(* CODESYS project xlh_ha_client_00_01.project
   Author: CODESYS Development GmbH
   Title: MQTT Client SL Example
   Company: CODESYS

Project tree, tasks and I/O mapping:
  Device : CODESYS Control for Raspberry Pi 64 SL, CODESYS, order no. 2302000009, version 4.12.0.0
    application app
      libraries: Standard, 3.5.18.0 (System); StringUtils, 3.5.20.0 (System); VisuDialogs, * (System); Web Socket Client SL, 1.12.0.0 (CODESYS); Net Base Services, * (3S - Smart Software Solutions GmbH); MQTT Client SL, 1.12.0.0 (CODESYS); Util, 3.5.21.0 (System); String Functions, * (CODESYS); SysTimeRtc, * (System); SysTime, 3.5.17.0 (System); CmpIecTask, * (System)
      task MainTask (cyclic, interval t#20ms, priority 1) calls LOCAL_TIME_AND_TIME_ZONE, TASK_INFO, io, MAIN
      program MAIN [ST]
      program io [ST]
      IoT/
        DEVICES/
          function block _100_FB_DEVICE [ST]: subscriber, publisher, pMqttClient, startup, sMqttTopicBase, newMessage, statusUpdate
          function block _200_FB_DEVICE_SHELLY_BASE [ST]: statusUpdate, startup, newMessage
          function block _202_FB_DEVICE_SHELLY_1PM_TEMP [ST]: newMessage
          interface IDevice
          interface IDeviceZigbee2Mqtt
          interface IDeviceShelly
          function block _201_FB_DEVICE_SHELLY_1PM_PLUG [ST]: publisher, newMessage
        MQTT_Client/
          function TERMINATE_STRING [ST]
          function block FB_MQTT_CLIENT [ST]: pMqttClient
          function GET_VALUE_FROM_MSG [ST]
          function GET_REAL_FROM_VALUE [ST]
          function GET_BOOL_FROM_VALUE [ST]
          function GET_INT_FROM_VALUE [ST]
          function GET_STRING_FROM_VALUE [ST]
        global variables GC
        program TASK_INFO [ST]
        program LOCAL_TIME_AND_TIME_ZONE [ST]
    SoftMotion General Axis Pool
    GPIOs_A_B : GPIOs A/B, CODESYS, version 4.18.0.0
        unmapped channels: digital inputs (GPIO0..GPIO31), digital outputs (GPIO0..GPIO31)
    Onewire
    Camera device
      <Empty>
    SPI
    I²C
  text list GlobalTextList
  5ce3da45-db07-42e7-a21c-a00fff4ed8f6|C:\Users\a.werner\Documents\background.jpg
*)

// Device/app/IoT/GC
{attribute 'qualified_only'}
VAR_GLOBAL CONSTANT
	//STRING_SIZE: INT := 255;
	STRING_SIZE_TOPIC: INT := 1024;
	STRING_SIZE_MESSAGE_RCV: INT := 2048;
END_VAR

// Device/app/IoT/LOCAL_TIME_AND_TIME_ZONE
PROGRAM LOCAL_TIME_AND_TIME_ZONE
VAR_OUTPUT
	stUTC_Timestamp : SysTime;
	stCTE_Timestamp : SysTime;
	stJoinedTimestamp : SysTime;
	stCombinedTimestamp : SysTime;
	uiYear : YEAR; (* 1970..2106 *)
    uiMonth : MONTH;
    uiDay : DAY;
    uiHour : UINT;
    uiMinute : UINT;
    uiSecond : UINT;
    uiMilliseconds : MILLISECOND;
    eWeekday : WEEKDAY;
    datDate : DATE;
    todTime : TIME_OF_DAY;
	eError : Util.ERROR;
	xLeapYear : BOOL;
END_VAR
VAR CONSTANT
    /// Coordinated Universal Time
    gc_tzTimeZoneUTC : TimeZone := (asgPeriod := [(sName:='UTC')]);

    /// Central Europe Time
    gc_tzTimeZoneCET : TimeZone :=
    (
        iBias := 60 (* T#1M => minutes *),
        asgPeriod := [
        ( (* (CEST -> CET) - Last Sunday in Oktober at 03:00:00.000 (CEST) *)
            sName:='CET',
            dtDate := (uiMonth := 10, eWeekday := WEEKDAY.SUNDAY, uiDay := 5, uiHour := 3)
        ),( (* (CET -> CEST) - Last Sunday in March at 02:00:00.000 (CET) *)
            sName := 'CEST',
            dtDate := (uiMonth := 3, eWeekday := WEEKDAY.SUNDAY, uiDay := 5, uiHour := 2),
            iBias := 60 (* T#1M => minutes *)
        )]
    );
END_VAR

SysTimeRtcHighResGet(pTimestamp := stUTC_Timestamp);
// Conversion from UTC timestamp (e.g. from SysTimeRtcHighResGet) to the current period and the local date and time related to the TimeZone parameter.
stCTE_Timestamp := Util.LocalDateTime(	tzTimeZone := gc_tzTimeZoneCET, 
										uliDateTime := stUTC_Timestamp,
										eErrorID => eError);

// Splitting a timestamp into the components of a point in time.
eError := Util.SplitDateTime(	uliDateTime := stCTE_Timestamp,
				uiYear => uiYear,
				uiMonth =>  uiMonth,
				uiDay => uiDay,
				uiHour => uiHour,
				uiMinute => uiMinute,
				uiSecond =>  uiSecond,
				uiMilliseconds => uiMilliseconds,
				eWeekday => eWeekday);

// Joining the components of a point in time to a timestamp (UTC). 
stJoinedTimestamp :=  Util.JoinDateTime( 	uiYear := uiYear,
									uiMonth :=  uiMonth,
									uiDay := uiDay,
									uiHour := uiHour,
									uiMinute := uiMinute,
									uiSecond :=  uiSecond,
									uiMilliseconds := uiMilliseconds);
									
// Separates a timestamp in its IEC data typed parts.
 Util.SeparateDateTime(	uliDateTime := stCTE_Timestamp,
    				eWeekDay => eWeekDay,
    				datDate => datDate,
    				todTime => todTime);
					
// Combines the IEC data typed parts to a timestamp.
stCombinedTimestamp := Util.CombineDateTime(	datDate := datDate, 
												todTime := todTime, 
												eErrorID => eError);
						
// Calculates the appropriate value of the WEEKDAY enum that matches the parameter datDate.
eWeekday := Util.DayOfWeek(	datDate := datDate, 
							eErrorID => eError);

// Checks whether the year (uiYear) passed represents a leap year.					
xLeapYear := Util.IsLeapYear(	uiYear := uiYear,
								eErrorID => eError);

END_PROGRAM

// Device/app/IoT/TASK_INFO
PROGRAM TASK_INFO
VAR
    Result: CmpIecTask.RTS_IEC_RESULT;
    hCurrentTask : CmpIecTask.RTS_IEC_HANDLE;
    pCurrentTaskInfo: POINTER TO Task_Info2;
    stCurrentTaskInfo: Task_Info2;
END_VAR
VAR_OUTPUT
	rCycleTime: REAL;
	rInterval: REAL;
	rCycleTimeUs: REAL;
	rJitterUs: REAL;
	rJitterOffsetInterwalUs: REAL;
END_VAR

// https://content.helpme-codesys.com/en/libs/CmpIecTask/Current/index.html
// https://forge.codesys.com/forge/talk/Engineering/thread/b7e9b2b353/
// https://medium.com/@sean.gongz/how-to-get-current-task-actual-cycle-time-in-codesys-267384bcd3b7

hCurrentTask := IecTaskGetCurrent(pResult:=ADR(Result));
pCurrentTaskInfo := IecTaskGetInfo3(hIecTask:=hCurrentTask, pResult:=ADR(Result));
stCurrentTaskInfo := pCurrentTaskInfo^;

rCycleTimeUs := TO_REAL(TO_DINT(stCurrentTaskInfo.dwInterval) + stCurrentTaskInfo.iJitter);
rInterval := TO_REAL(stCurrentTaskInfo.dwInterval);
rJitterUs := TO_REAL(stCurrentTaskInfo.iJitter);
rJitterOffsetInterwalUs := rInterval + rJitterUs;
rCycleTime := rCycleTimeUs / 1000000.0;

END_PROGRAM

// Device/app/io
PROGRAM io
VAR_INPUT
	fbShellyPlug1: _201_FB_DEVICE_SHELLY_1PM_PLUG;
	fbShellyPlug2: _201_FB_DEVICE_SHELLY_1PM_PLUG;
	fbShellyPm1: _202_FB_DEVICE_SHELLY_1PM_TEMP;
END_VAR
VAR
	_bStartup: BOOL := TRUE;
	_aIoClients: ARRAY [0..(iNR_OF_IO_CLIENTS-1)] OF POINTER TO _100_FB_DEVICE;
	_fbMqttClient: FB_MQTT_CLIENT;
	_iI: INT;
	//
	_bDummy: BOOL;
END_VAR
VAR CONSTANT
	iNR_OF_IO_CLIENTS: INT := 20;
END_VAR

IF _bStartup THEN
	_bStartup := FALSE;
	
	fbShellyPlug1.sMqttTopicBase := 'shellyplug-81';
	fbShellyPlug2.sMqttTopicBase := 'shellyplug-82';
	fbShellyPm1.sMqttTopicBase := 'shellyplus-51';
	
	_aIoClients[_iI] := ADR(fbShellyPlug1); _iI := _iI + 1;
	_aIoClients[_iI] := ADR(fbShellyPlug2); _iI := _iI + 1;
	_aIoClients[_iI] := ADR(fbShellyPm1); _iI := _iI + 1;
	
	FOR _iI := 0 TO (iNR_OF_IO_CLIENTS-1) BY 1 DO
		IF (_aIoClients[_iI] > 16#0) THEN
			_aIoClients[_iI]^.pMqttClient := ADR(_fbMqttClient);
			_aIoClients[_iI]^.startup();	
		END_IF
	END_FOR	
	
	_fbMqttClient.bEnable := TRUE;
END_IF

_fbMqttClient();

FOR _iI := 0 TO (iNR_OF_IO_CLIENTS-1) BY 1 DO
	IF (_aIoClients[_iI] >16#0) THEN
		_aIoClients[_iI]^();	
	END_IF
END_FOR

_bDummy := _fbMqttClient.bConnected;

END_PROGRAM

// Device/app/IoT/DEVICES/_201_FB_DEVICE_SHELLY_1PM_PLUG
FUNCTION_BLOCK _201_FB_DEVICE_SHELLY_1PM_PLUG EXTENDS _200_FB_DEVICE_SHELLY_BASE
VAR_INPUT
	bRelais: BOOL;
END_VAR
VAR_OUTPUT
	bRelaisState: BOOL;
	rVoltage: REAL;
	rCurrent: REAL;
	rPower: REAL;
END_VAR
VAR
	//
	_fbRtRelais: R_TRIG;
	_fbFtRelais: F_tRIG;
	_fbTonDiffRelaisState: TON;
END_VAR
VAR CONSTANT
	_tACTION_TIME_NOT_EQUAL: TIME := T#500MS;
END_VAR

SUPER^();

METHOD publisher : BOOL
VAR_INPUT
END_VAR

VAR
	bPublish: BOOL;
END_VAR
THIS^._fbTonDiffRelaisState(IN:=((THIS^.bRelais <> THIS^.bRelaisState) AND NOT _fbTonDiffRelaisState.Q), PT:=THIS^._tACTION_TIME_NOT_EQUAL);
THIS^._fbRtRelais(CLK:=THIS^.bRelais);
THIS^._fbFtRelais(CLK:=THIS^.bRelais);
bPublish := _fbTonDiffRelaisState.Q OR _fbRtRelais.Q OR _fbFtRelais.Q;

IF bPublish THEN
	THIS^._fbMqttPublisher.xExecute := TRUE;
	THIS^._sPublishMessage := '{"id":1, "src":"';
	THIS^._sPublishMessage := CONCAT(THIS^._sPublishMessage, THIS^._sMqttTopicBase);
	THIS^._sPublishMessage := CONCAT(THIS^._sPublishMessage, '/relais", "method":"Switch.Set", "params":{"id":0, "on":');
	IF THIS^.bRelais THEN
		THIS^._sPublishMessage := CONCAT(THIS^._sPublishMessage, 'true}}');
	ELSE
		THIS^._sPublishMessage := CONCAT(THIS^._sPublishMessage, 'false}}');
	END_IF
END_IF

SUPER^.publisher();

// '{"id":1, "src":"shellyplus-51/status", "method":"Shelly.GetStatus"}'
//{"id":1, "src":"shellyplus-51/relais", "method":"Switch.Set", "params":{"id":0, "on":true}}
END_METHOD

METHOD newMessage : BOOL
VAR_INPUT
	
END_VAR
VAR

	
END_VAR
SUPER^.newMessage();
IF (_fbMqttSubscriber.wsLastTopic = _wsMqttTopicEvent) OR
   (_fbMqttSubscriber.wsLastTopic = _wsMqttTopicStatus) THEN
	bRelaisState := GET_BOOL_FROM_VALUE(bRelaisState, GET_VALUE_FROM_MSG('output', ADR(_sSubscribedMessage)));
	rVoltage := GET_REAL_FROM_VALUE(rVoltage, GET_VALUE_FROM_MSG('voltage', ADR(_sSubscribedMessage)));
	rCurrent := GET_REAL_FROM_VALUE(rCurrent, GET_VALUE_FROM_MSG('current', ADR(_sSubscribedMessage)));
	rPower := GET_REAL_FROM_VALUE(rPower, GET_VALUE_FROM_MSG('apower', ADR(_sSubscribedMessage)));
		
END_IF
IF (_fbMqttSubscriber.wsLastTopic = _wsMqttTopicStatus) THEN
	sSsid := GET_STRING_FROM_VALUE(sSsid, GET_VALUE_FROM_MSG('ssid', ADR(_sSubscribedMessage)));
	sMacId := GET_STRING_FROM_VALUE(sSsid, GET_VALUE_FROM_MSG('bssid', ADR(_sSubscribedMessage)));	
END_IF
END_METHOD

END_FUNCTION_BLOCK

// Device/app/IoT/DEVICES/_200_FB_DEVICE_SHELLY_BASE
FUNCTION_BLOCK _200_FB_DEVICE_SHELLY_BASE EXTENDS _100_FB_DEVICE IMPLEMENTS IDeviceShelly
VAR_INPUT
END_VAR
VAR_OUTPUT
	rTemperaturePcb: REAL;
	sSsid: STRING(255);
	sMacId: STRING(255);
	iRssi: INT;
END_VAR
VAR
	//
	_wsMqttTopicEvent: WSTRING(GC.STRING_SIZE_TOPIC) := "shellyplus-51/status/rpc";
	_wsMqttTopicStatus: WSTRING(GC.STRING_SIZE_TOPIC) := "shellyplus-51/status/rpc";
	_rTimer: REAL := 0.0;
END_VAR
VAR CONSTANT
	_rREFRESH_TIME: REAL := 300.0;
END_VAR

SUPER^();

_rTimer := LIMIT(0.0, _rTimer + TASK_INFO.rCycleTime, 99999.0);
IF _rTimer >= _rREFRESH_TIME THEN
	_rTimer := 0.0;
	statusUpdate();
END_IF

METHOD statusUpdate : BOOL
VAR_INPUT
END_VAR

VAR
END_VAR
SUPER^.statusUpdate();

THIS^._fbMqttPublisher.xExecute := TRUE;
THIS^._sPublishMessage := '{"id":1, "src":"';
THIS^._sPublishMessage := CONCAT(THIS^._sPublishMessage, THIS^._sMqttTopicBase);
THIS^._sPublishMessage := CONCAT(THIS^._sPublishMessage, '/status", "method":"Shelly.GetStatus"}');

// '{"id":1, "src":"shellyplus-51/status", "method":"Shelly.GetStatus"}'
END_METHOD

METHOD startup : BOOL
VAR_INPUT
END_VAR

VAR
END_VAR
SUPER^.startup();

_wsMqttTopicEvent := "";
Stu.StrConcatW(pstFrom:=ADR(_wsMqttTopicBase), pstTo:=ADR(_wsMqttTopicEvent), iBufferSize:=GC.STRING_SIZE_TOPIC);
Stu.StrConcatW(pstFrom:=ADR("/events/rpc"), pstTo:=ADR(_wsMqttTopicEvent), iBufferSize:=GC.STRING_SIZE_TOPIC);
		
_wsMqttTopicStatus := "";
Stu.StrConcatW(pstFrom:=ADR(_wsMqttTopicBase), pstTo:=ADR(_wsMqttTopicStatus), iBufferSize:=GC.STRING_SIZE_TOPIC);
Stu.StrConcatW(pstFrom:=ADR("/status/rpc"), pstTo:=ADR(_wsMqttTopicStatus), iBufferSize:=GC.STRING_SIZE_TOPIC);
END_METHOD

METHOD newMessage : BOOL
VAR_INPUT
	
END_VAR
VAR

	
END_VAR
SUPER^.newMessage();
IF (_fbMqttSubscriber.wsLastTopic = _wsMqttTopicEvent) OR
   (_fbMqttSubscriber.wsLastTopic = _wsMqttTopicStatus) THEN
   rTemperaturePcb := GET_REAL_FROM_VALUE(rTemperaturePcb, GET_VALUE_FROM_MSG('temperature":{"tC', ADR(_sSubscribedMessage)));
	iRssi := GET_INT_FROM_VALUE(iRssi, GET_VALUE_FROM_MSG('rssi', ADR(_sSubscribedMessage)));	
END_IF
IF (_fbMqttSubscriber.wsLastTopic = _wsMqttTopicStatus) THEN
	sSsid := GET_STRING_FROM_VALUE(sSsid, GET_VALUE_FROM_MSG('ssid', ADR(_sSubscribedMessage)));
	sMacId := GET_STRING_FROM_VALUE(sSsid, GET_VALUE_FROM_MSG('bssid', ADR(_sSubscribedMessage)));	
END_IF
END_METHOD

END_FUNCTION_BLOCK

// Device/app/IoT/DEVICES/_100_FB_DEVICE
FUNCTION_BLOCK _100_FB_DEVICE IMPLEMENTS IDevice
VAR
	_pMqttClient: POINTER TO FB_MQTT_CLIENT;
	_wsMqttTopicBase: WSTRING(GC.STRING_SIZE_TOPIC);
	_sMqttTopicBase: STRING(255);
	//
	_fbRtMqttClientConnected: R_TRIG;
	_fbFtMqttClientConnected: F_TRIG;
	_fbRtMqttSubscriberActive: R_TRIG;
	_fbFtMqttSubscriberActive: F_TRIG;
	_fbRtError: R_TRIG;
	_fbTonConnect: TON;
	_fbTonDisconnect: TON;
	_fbMqttSubscriber : MQTT.MQTTSubscribe;
	_wsSubcribedTopicFilter : WSTRING(GC.STRING_SIZE_TOPIC);
	_sSubscribedMessage : STRING(GC.STRING_SIZE_MESSAGE_RCV);	
	_fbMqttPublisher : MQTT.MQTTPublish;
	_wsPublishTopic : WSTRING(GC.STRING_SIZE_TOPIC);
	_sPublishMessage : STRING(255);
	//
	_todMessageUpdate: TIME_OF_DAY;
	//
	_bDummy: BOOL;
	_iDummyCtr: INT;
	_sDummy: STRING(GC.STRING_SIZE_MESSAGE_RCV);
	_wsDummy: WSTRING(GC.STRING_SIZE_TOPIC);
END_VAR

(*
Optimierung:
- Queue für Verarbeitung ausgehender Nachrichten
- Interface
- REAL mit LReal ersetzen
*)

THIS^.subscriber();
THIS^.publisher();

METHOD subscriber : BOOL
VAR_INPUT
END_VAR
THIS^._fbRtMqttClientConnected(CLK:=THIS^._pMqttClient^.bConnected);
THIS^._fbFtMqttClientConnected(CLK:=THIS^._pMqttClient^.bConnected);
THIS^._fbRtError(CLK:=THIS^._pMqttClient^.bError);
IF THIS^._fbRtMqttClientConnected.Q THEN
	THIS^._fbMqttSubscriber.xEnable := TRUE;
END_IF
IF THIS^._fbRtError.Q OR THIS^._fbFtMqttClientConnected.Q THEN
	THIS^._fbMqttSubscriber.xEnable := FALSE;
END_IF
THIS^._fbTonDisconnect.IN := THIS^._pMqttClient^.bConnected AND THIS^._fbMqttSubscriber.xEnable AND NOT THIS^._fbMqttSubscriber.xBusy;
THIS^._fbTonDisconnect(PT:=T#3000MS);
IF THIS^._fbTonDisconnect.Q THEN
	THIS^._fbMqttSubscriber.xEnable := FALSE;
END_IF
THIS^._fbTonConnect.IN := THIS^._pMqttClient^.bConnected AND NOT THIS^._fbMqttSubscriber.xEnable;
THIS^._fbTonConnect(PT:=T#500MS);
IF THIS^._fbTonConnect.Q THEN
	THIS^._fbMqttSubscriber.xEnable := TRUE;
END_IF

THIS^._fbMqttSubscriber(mqttClient:=THIS^._pMqttClient^.fbMqttClient,
				wsTopicFilter:=THIS^._wsSubcribedTopicFilter,
		        pbPayload:=ADR(THIS^._sSubscribedMessage),
				udiMaxPayloadSize:=SIZEOF(THIS^._sSubscribedMessage));
TERMINATE_STRING(psIn:=ADR(THIS^._sSubscribedMessage), THIS^._fbMqttSubscriber.udiPayloadSize);

IF THIS^._fbMqttSubscriber.xReceived THEN
	THIS^.newMessage();
END_IF 

THIS^._fbRtMqttSubscriberActive(CLK:=THIS^._fbMqttSubscriber.xSubscribeActive);
THIS^._fbFtMqttSubscriberActive(CLK:=THIS^._fbMqttSubscriber.xSubscribeActive);
IF THIS^._fbRtMqttSubscriberActive.Q THEN
	THIS^.statusUpdate();
END_IF
			
_bDummy := THIS^._fbMqttSubscriber.xEnable;				
_bDummy := THIS^._fbMqttSubscriber.xDone;
_bDummy := THIS^._fbMqttSubscriber.xBusy;
_bDummy := THIS^._fbMqttSubscriber.xError;
_bDummy := THIS^._fbMqttSubscriber.xSubscribeActive;
_wsDummy := THIS^._fbMqttSubscriber.wsLastTopic;
_sDummy := THIS^._sSubscribedMessage;
END_METHOD

METHOD publisher : BOOL
VAR_INPUT
END_VAR
THIS^._fbMqttPublisher(mqttClient:=_pMqttClient^.fbMqttClient, 	 
                       wsTopicName:=_wsPublishTopic,
                       udiTimeOut:=10000,
                       pbPayload:=ADR(_sPublishMessage),
	                   udiPayloadSize:=DINT_TO_UDINT(Stu.StrLenA(ADR(_sPublishMessage))));

(*
// Send Counter
IF _fbMqttPublisher.xBusy THEN
	_iDummyCtr := _iDummyCtr + 1;
END_IF
*)

THIS^._fbMqttPublisher.xExecute := FALSE;   

_bDummy := _fbMqttPublisher.xDone;
_bDummy := _fbMqttPublisher.xBusy;
_bDummy := _fbMqttPublisher.xError;
_wsDummy := _wsPublishTopic;
_sDummy := _sPublishMessage;
END_METHOD

PROPERTY pMqttClient : POINTER TO FB_MQTT_CLIENT
GET
pMqttClient := THIS^._pMqttClient;
END_GET
SET
THIS^._pMqttClient := pMqttClient;
END_SET
END_PROPERTY

METHOD startup : BOOL
VAR_INPUT
END_VAR

VAR
END_VAR
_wsMqttTopicBase := STRING_TO_WSTRING(_sMqttTopicBase);

_wsPublishTopic := "";
Stu.StrConcatW(pstFrom:=ADR(_wsMqttTopicBase), pstTo:=ADR(_wsPublishTopic), iBufferSize:=GC.STRING_SIZE_TOPIC);
Stu.StrConcatW(pstFrom:=ADR("/rpc"), pstTo:=ADR(_wsPublishTopic), iBufferSize:=GC.STRING_SIZE_TOPIC);

_wsSubcribedTopicFilter := "";
Stu.StrConcatW(pstFrom:=ADR(_wsMqttTopicBase), pstTo:=ADR(_wsSubcribedTopicFilter), iBufferSize:=GC.STRING_SIZE_TOPIC);
Stu.StrConcatW(pstFrom:=ADR("/#"), pstTo:=ADR(_wsSubcribedTopicFilter), iBufferSize:=GC.STRING_SIZE_TOPIC);
END_METHOD

PROPERTY PUBLIC sMqttTopicBase : STRING(255)
SET
THIS^._sMqttTopicBase := sMqttTopicBase;
END_SET
GET
sMqttTopicBase := THIS^._sMqttTopicBase;
END_GET
END_PROPERTY

METHOD newMessage : BOOL
VAR_INPUT
	
END_VAR
VAR

	
END_VAR
THIS^._todMessageUpdate := LOCAL_TIME_AND_TIME_ZONE.todTime;
END_METHOD

METHOD statusUpdate : BOOL
VAR_INPUT
END_VAR

VAR
END_VAR
END_METHOD

END_FUNCTION_BLOCK

// Device/app/IoT/DEVICES/IDevice
INTERFACE IDevice

END_INTERFACE

// Device/app/IoT/MQTT_Client/FB_MQTT_CLIENT
FUNCTION_BLOCK FB_MQTT_CLIENT
VAR_INPUT
	bEnable: BOOL;
	sHostname: STRING(255) := 'localhost';	
	sClientId: STRING(255) := 'xLH_mqtt_codesys';	
END_VAR
VAR_OUTPUT
	bConnected: BOOL;
	bError: BOOL;
	fbMqttClient : MQTT.MQTTClient := (uiPort:=1883, eMQTTVersion:=MQTT.MQTT_VERSION.V3_1_1, eCommunicationMode:= MQTT.COMMUNICATION_MODE.TCP);
END_VAR
VAR
	_refMqttClient: REFERENCE TO MQTT.MQTTClient;
	_bStartup: BOOL := TRUE;
END_VAR

IF _bStartup THEN
	_bStartup := FALSE;
	_refMqttClient REF= fbMqttClient;
END_IF
fbMqttClient.xEnable := bEnable AND NOT fbMqttClient.xError;
fbMqttClient.sClientId := sClientId;
fbMqttClient(sHostname:=sHostname);
bConnected := fbMqttClient.xConnectedToBroker;
bError := fbMqttClient.xError;

PROPERTY pMqttClient : POINTER TO FB_MQTT_CLIENT
GET
pMqttClient := ADR(THIS^.fbMqttClient);
END_GET
END_PROPERTY

END_FUNCTION_BLOCK

// Device/app/IoT/MQTT_Client/TERMINATE_STRING
// Terminates the STRING psIn at position udiLength
FUNCTION TERMINATE_STRING : BOOL
VAR_INPUT
	psIn : POINTER TO BYTE; // Pointer to STRING
	udiLength : UDINT; // Length of psIn
END_VAR
VAR
END_VAR

psIn[udiLength] := 0;
TERMINATE_STRING := TRUE;

END_FUNCTION

// Device/app/IoT/DEVICES/IDeviceShelly
INTERFACE IDeviceShelly

END_INTERFACE

// Device/app/IoT/MQTT_Client/GET_REAL_FROM_VALUE
FUNCTION GET_REAL_FROM_VALUE: REAL;
VAR_INPUT
	rValue: REAL;
	sValue: STRING(255);
END_VAR

IF sValue <> '' THEN
	rValue := STRING_TO_REAL(sValue);
END_IF
GET_REAL_FROM_VALUE := rValue;

END_FUNCTION

// Device/app/IoT/MQTT_Client/GET_VALUE_FROM_MSG
FUNCTION GET_VALUE_FROM_MSG: STRING(255)
VAR_INPUT
	sKey: STRING(255);
	pSubscribedMessage: POINTER TO STRING(GC.STRING_SIZE_MESSAGE_RCV);
END_VAR
VAR
	iStrFindPos1: INT;
	iStrFindPos2: INT;
	sMessage : STRING(255);
	sValue : STRING(255);
END_VAR

sKey := CONCAT(CONCAT('"', sKey), '":'); 		

iStrFindPos1 := MAX(0, Stu.StrFindA(pst1:=pSubscribedMessage, pst2:=ADR(sKey), uiSearchStart:=0));
Stu.StrCpyA(pBuffer:=ADR(sMessage), 
			iBufferSize:=SIZEOF(sMessage)-50, 
			pStr:=pSubscribedMessage+INT_TO_DWORD(iStrFindPos1));  

iStrFindPos1 := MAX(0, Stu.StrFindA(pst1:=ADR(sMessage), 
                                    pst2:=ADR(':'), 
                                    uiSearchStart:=INT_TO_UINT(MAX(0, LEN(sKey)-1))));		 
iStrFindPos2 := MAX(0, Stu.StrFindA(pst1:=ADR(sMessage), 
                                    pst2:=ADR(','), 
                                    uiSearchStart:=INT_TO_UINT(MAX(0, LEN(sKey)))));		
IF iStrFindPos2 = 0 THEN
	iStrFindPos2 := MAX(0, Stu.StrFindA(pst1:=ADR(sMessage), 
                                    pst2:=ADR('}'), 
                                    uiSearchStart:=INT_TO_UINT(MAX(0, LEN(sKey)))));
END_IF
// Falls das Property nicht vorhanden ist, keine Aenderung
IF (iStrFindPos1 <> 0) AND (iStrFindPos2 <> 0) THEN
	sValue := MID(sMessage, iStrFindPos2-iStrFindPos1-1, iStrFindPos1+1);
	// bei einem String sind die " zu enternen
	IF LEFT(sMessage, 1) = '"' THEN
		sValue := MID(sValue, LEN(sValue)-2, 2);
	END_IF
ELSE
	sValue := '';
END_IF
		
(*
sValue := '';
sValue := CONCAT(sValue, INT_TO_STRING(iStrFindPos1));
sValue := CONCAT(sValue, ' | ');
sValue := CONCAT(sValue, INT_TO_STRING(iStrFindPos2));
sValue := CONCAT(sValue, ' | ');
sValue := CONCAT(sValue, sMessage);
*)

GET_VALUE_FROM_MSG := sValue;

END_FUNCTION

// Device/app/IoT/MQTT_Client/GET_INT_FROM_VALUE
FUNCTION GET_INT_FROM_VALUE: INT;
VAR_INPUT
	iValue: int;
	sValue: STRING(255);
END_VAR

IF sValue <> '' THEN
	iValue := STRING_TO_INT(sValue);
END_IF
GET_INT_FROM_VALUE := iValue;

END_FUNCTION

// Device/app/IoT/MQTT_Client/GET_STRING_FROM_VALUE
FUNCTION GET_STRING_FROM_VALUE: STRING(255);
VAR_INPUT
	_sValue: STRING(255);
	sValue: STRING(255);
END_VAR

IF sValue <> '' THEN
	_sValue := sValue;
END_IF
GET_STRING_FROM_VALUE := _sValue;

END_FUNCTION

// Device/app/IoT/MQTT_Client/GET_BOOL_FROM_VALUE
FUNCTION GET_BOOL_FROM_VALUE: BOOL;
VAR_INPUT
	bValue: BOOL;
	sValue: STRING(255);
END_VAR

IF sValue <> '' THEN
	bValue := (sValue = 'true');
END_IF
GET_BOOL_FROM_VALUE := bValue;

END_FUNCTION

// Device/app/IoT/DEVICES/_202_FB_DEVICE_SHELLY_1PM_TEMP
FUNCTION_BLOCK _202_FB_DEVICE_SHELLY_1PM_TEMP EXTENDS _201_FB_DEVICE_SHELLY_1PM_PLUG
VAR_OUTPUT
	rTemperature1: REAL;
	rTemperature2: REAL;
	rTemperature3: REAL;
END_VAR

SUPER^();

METHOD newMessage : BOOL
VAR_INPUT
	
END_VAR
VAR

	
END_VAR
SUPER^.newMessage();
IF (_fbMqttSubscriber.wsLastTopic = _wsMqttTopicEvent) OR
   (_fbMqttSubscriber.wsLastTopic = _wsMqttTopicStatus) THEN
	rTemperature1 := GET_REAL_FROM_VALUE(rTemperature1, GET_VALUE_FROM_MSG('temperature:100":{"id": 100,"tC', ADR(_sSubscribedMessage)));
	rTemperature1 := GET_REAL_FROM_VALUE(rTemperature1, GET_VALUE_FROM_MSG('temperature:100":{"tC', ADR(_sSubscribedMessage)));
	rTemperature2 := GET_REAL_FROM_VALUE(rTemperature2, GET_VALUE_FROM_MSG('temperature:101":{"id": 101,"tC', ADR(_sSubscribedMessage)));
	rTemperature2 := GET_REAL_FROM_VALUE(rTemperature2, GET_VALUE_FROM_MSG('temperature:101":{"tC', ADR(_sSubscribedMessage)));
	rTemperature3 := GET_REAL_FROM_VALUE(rTemperature3, GET_VALUE_FROM_MSG('temperature:102":{"id": 102,"tC', ADR(_sSubscribedMessage)));
	rTemperature3 := GET_REAL_FROM_VALUE(rTemperature3, GET_VALUE_FROM_MSG('temperature:102":{"tC', ADR(_sSubscribedMessage)));
END_IF
END_METHOD

END_FUNCTION_BLOCK

// Device/app/MAIN
PROGRAM MAIN
VAR
END_VAR

(*
IP Shelly Accesspoint: 192.168.33.1
IP Shelly ABB-Technikerschule: 172.16.23.118
*)

END_PROGRAM

// Device/app/IoT/DEVICES/IDeviceZigbee2Mqtt
INTERFACE IDeviceZigbee2Mqtt

END_INTERFACE
